FUNCTION_BLOCK myVeryFirstTcoContext EXTENDS TcoCore.TcoContext
VAR
	{attribute addProperty Name "<#My very first DATAMAN#>"}
	myVeryFirstDataman : TcoCognexVision.TcoDataman_v_5_x_x(THIS^);
	{attribute addProperty Name "<#My very first INSIGHT#>"}
	myVeryFirstInsight : TcoCognexVision.TcoInsight_v_5_x_x(THIS^);

	

	{attribute addProperty Name "<#Cognex Designer#>"}
	designer : TcoCognexVision.TcoDesigner_v_2_x_x(THIS^);
	
	{attribute addProperty Name "<#Project Specific Data#>"}
    _specificData : ProjectSpecificData(THIS^);
	


END_VAR

(*~
	<docu>
		<summary>
			Main method of the TcoContext. This is the entry point of any control logic that belongs to this context. 
			The call of this method is ensured by calling the <c>InstanceName.Run()</c> method, and it must not be called explicitly.
			This method is abstract, and it must be overridden in derived block.
		</summary>
	</docu>
~*)
METHOD PROTECTED  Main

VAR
	
END_VAR
myVeryFirstDataman(inoIoData:= GVL.myVeryFirstDatamanGVL);
myVeryFirstDataman.Service();

myVeryFirstInsight.Config.UserDataSize := eTcoInsightUserDataSize_v_5_x_x.USER_DATA_128B;
myVeryFirstInsight.Config.ResultDataSize := eTcoInsightResultDataSize_v_5_x_x.RESULT_DATA_128B;
myVeryFirstInsight(inoIoData:= GVL.myVeryFirstInsightGVL);
myVeryFirstInsight.Service();
myVeryFirstDataman.Read();
myVeryFirstDataman.GetResultAsString(0,myVeryFirstDataman.Status.SignalStatus.ResultLength);




designer(inoData:=_specificData );
designer.Service();
END_METHOD

END_FUNCTION_BLOCK

(* stored: Version 1.1.0.1, ProductVersion 3.1.4024.12
   POU myVeryFirstTcoContext: Id {6a4dbc2d-6b21-0fcb-2bc4-0055ab5a286d}, SpecialFunc None
   Method Main: Id {62509618-e1c7-0fff-1ad6-21ea3ba2bca5} *)
